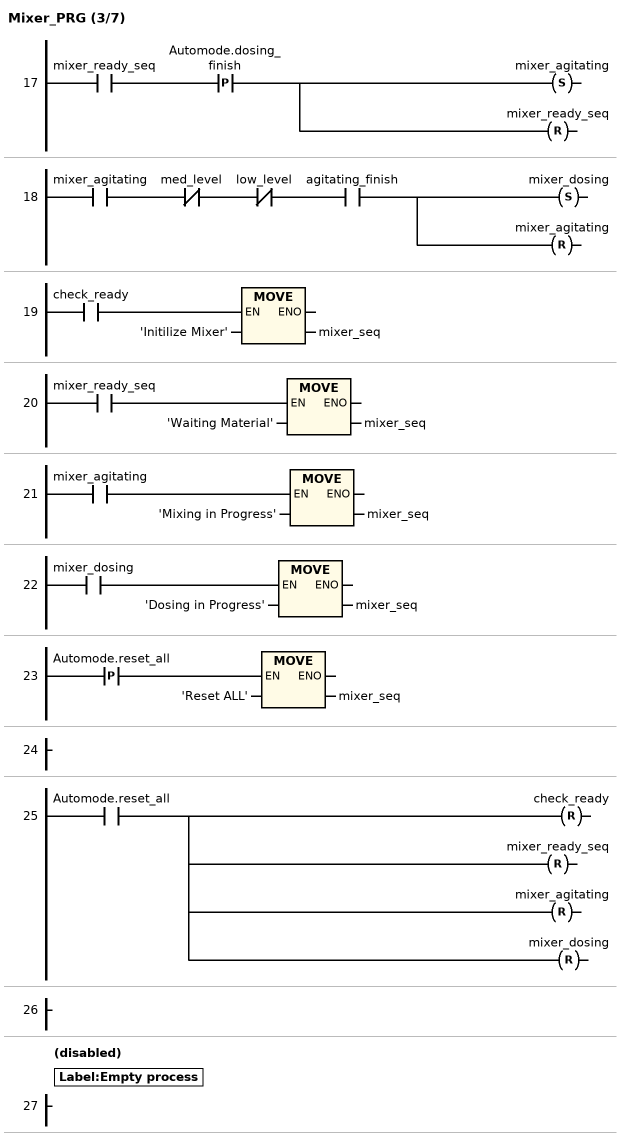
// NETWORK 17
_rt10(CLK := Automode.dosing_finish);
_w3 := mixer_ready_seq AND _rt10.Q;
mixer_agitating S= _w3;
mixer_ready_seq R= _w3;

// NETWORK 18
_w4 := mixer_agitating AND NOT med_level AND NOT low_level AND agitating_finish;
mixer_dosing S= _w4;
mixer_agitating R= _w4;

// NETWORK 19
IF check_ready THEN mixer_seq := 'Initilize Mixer'; END_IF

// NETWORK 20
IF mixer_ready_seq THEN mixer_seq := 'Waiting Material'; END_IF

// NETWORK 21
IF mixer_agitating THEN mixer_seq := 'Mixing in Progress'; END_IF

// NETWORK 22
IF mixer_dosing THEN mixer_seq := 'Dosing in Progress'; END_IF

// NETWORK 23
_rt11(CLK := Automode.reset_all);
IF _rt11.Q THEN mixer_seq := 'Reset ALL'; END_IF

// NETWORK 24

// NETWORK 25
check_ready R= Automode.reset_all;
mixer_ready_seq R= Automode.reset_all;
mixer_agitating R= Automode.reset_all;
mixer_dosing R= Automode.reset_all;

// NETWORK 26

// NETWORK 27 (disabled)
// label: Label:Empty process

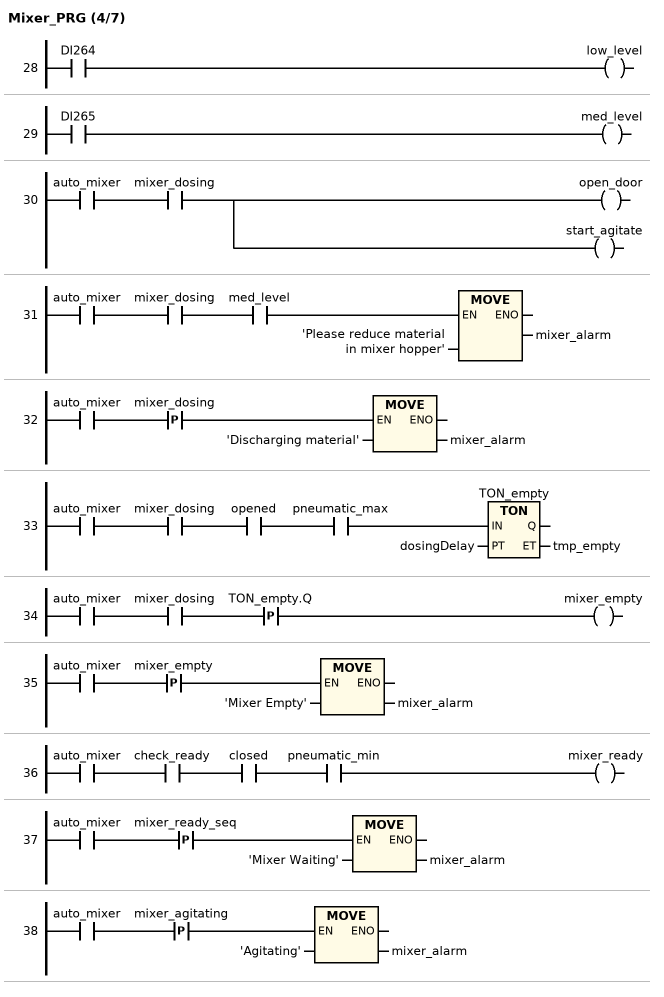
// NETWORK 28
low_level := DI264;

// NETWORK 29
med_level := DI265;

// NETWORK 30
_w5 := auto_mixer AND mixer_dosing;
open_door := _w5;
start_agitate := _w5;

// NETWORK 31
IF auto_mixer AND mixer_dosing AND med_level THEN mixer_alarm := 'Please reduce material in mixer hopper'; END_IF

// NETWORK 32
_rt12(CLK := mixer_dosing);
IF auto_mixer AND _rt12.Q THEN mixer_alarm := 'Discharging material'; END_IF

// NETWORK 33
TON_empty(IN := auto_mixer AND mixer_dosing AND opened AND pneumatic_max, PT := dosingDelay, ET => tmp_empty); // TON

// NETWORK 34
_rt13(CLK := TON_empty.Q);
mixer_empty := auto_mixer AND mixer_dosing AND _rt13.Q;

// NETWORK 35
_rt14(CLK := mixer_empty);
IF auto_mixer AND _rt14.Q THEN mixer_alarm := 'Mixer Empty'; END_IF

// NETWORK 36
mixer_ready := auto_mixer AND check_ready AND closed AND pneumatic_min;

// NETWORK 37
_rt15(CLK := mixer_ready_seq);
IF auto_mixer AND _rt15.Q THEN mixer_alarm := 'Mixer Waiting'; END_IF

// NETWORK 38
_rt16(CLK := mixer_agitating);
IF auto_mixer AND _rt16.Q THEN mixer_alarm := 'Agitating'; END_IF

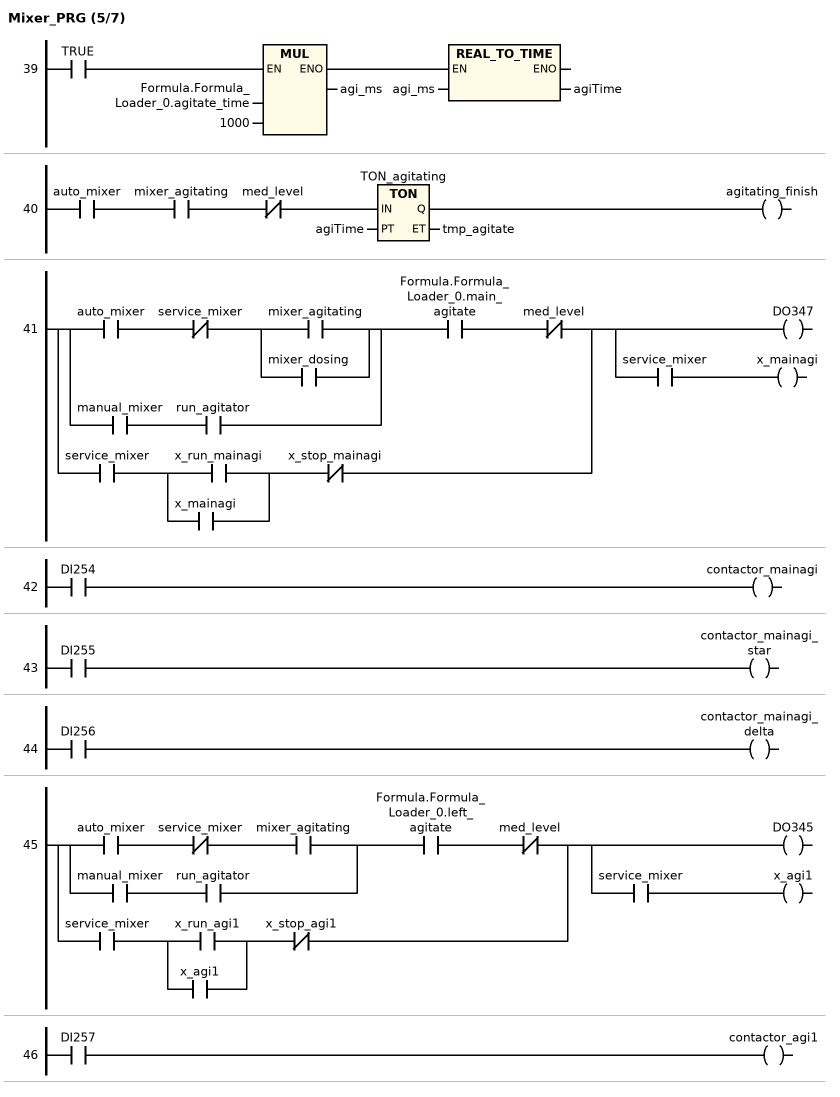
// NETWORK 39
agi_ms := Formula.Formula_Loader_0.agitate_time * 1000;
agiTime := REAL_TO_TIME(agi_ms);

// NETWORK 40
TON_agitating(IN := auto_mixer AND mixer_agitating AND NOT med_level, PT := agiTime, ET => tmp_agitate); // TON
agitating_finish := TON_agitating.Q;

// NETWORK 41
_w6 := (auto_mixer AND NOT service_mixer AND (mixer_agitating OR mixer_dosing) OR manual_mixer AND run_agitator) AND Formula.Formula_Loader_0.main_agitate AND NOT med_level OR service_mixer AND (x_run_mainagi OR x_mainagi) AND NOT x_stop_mainagi;
DO347 := _w6;
x_mainagi := _w6 AND service_mixer;

// NETWORK 42
contactor_mainagi := DI254;

// NETWORK 43
contactor_mainagi_star := DI255;

// NETWORK 44
contactor_mainagi_delta := DI256;

// NETWORK 45
_w7 := (auto_mixer AND NOT service_mixer AND mixer_agitating OR manual_mixer AND run_agitator) AND Formula.Formula_Loader_0.left_agitate AND NOT med_level OR service_mixer AND (x_run_agi1 OR x_agi1) AND NOT x_stop_agi1;
DO345 := _w7;
x_agi1 := _w7 AND service_mixer;

// NETWORK 46
contactor_agi1 := DI257;

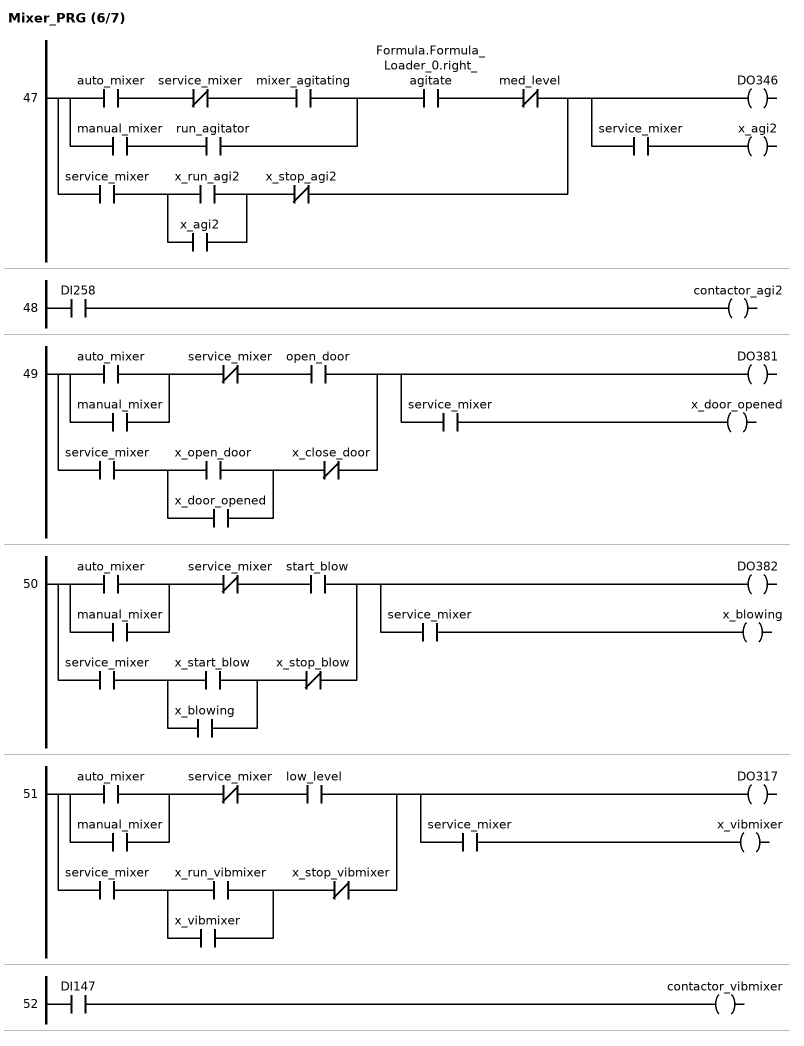
// NETWORK 47
_w8 := (auto_mixer AND NOT service_mixer AND mixer_agitating OR manual_mixer AND run_agitator) AND Formula.Formula_Loader_0.right_agitate AND NOT med_level OR service_mixer AND (x_run_agi2 OR x_agi2) AND NOT x_stop_agi2;
DO346 := _w8;
x_agi2 := _w8 AND service_mixer;

// NETWORK 48
contactor_agi2 := DI258;

// NETWORK 49
_w9 := (auto_mixer OR manual_mixer) AND NOT service_mixer AND open_door OR service_mixer AND (x_open_door OR x_door_opened) AND NOT x_close_door;
DO381 := _w9;
x_door_opened := _w9 AND service_mixer;

// NETWORK 50
_w10 := (auto_mixer OR manual_mixer) AND NOT service_mixer AND start_blow OR service_mixer AND (x_start_blow OR x_blowing) AND NOT x_stop_blow;
DO382 := _w10;
x_blowing := _w10 AND service_mixer;

// NETWORK 51
_w11 := (auto_mixer OR manual_mixer) AND NOT service_mixer AND low_level OR service_mixer AND (x_run_vibmixer OR x_vibmixer) AND NOT x_stop_vibmixer;
DO317 := _w11;
x_vibmixer := _w11 AND service_mixer;

// NETWORK 52
contactor_vibmixer := DI147;

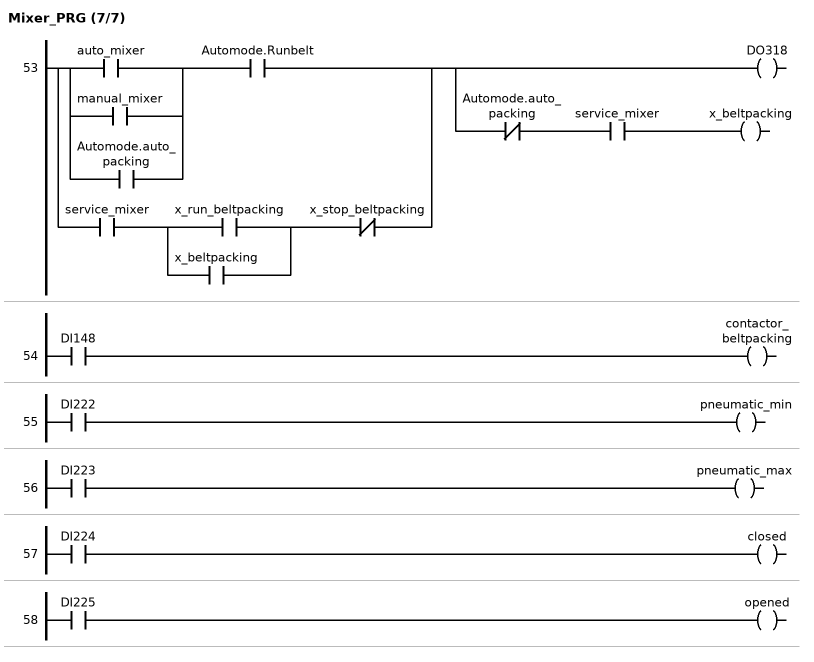
// NETWORK 53
_w12 := (auto_mixer OR manual_mixer OR Automode.auto_packing) AND Automode.Runbelt OR service_mixer AND (x_run_beltpacking OR x_beltpacking) AND NOT x_stop_beltpacking;
DO318 := _w12;
x_beltpacking := _w12 AND NOT Automode.auto_packing AND service_mixer;

// NETWORK 54
contactor_beltpacking := DI148;

// NETWORK 55
pneumatic_min := DI222;

// NETWORK 56
pneumatic_max := DI223;

// NETWORK 57
closed := DI224;

// NETWORK 58
opened := DI225;

END_PROGRAM

// Device/Application/LimeSand
PROGRAM LimeSand
VAR
	auto_lime: BOOL;
	manual_lime: BOOL;
	manual_dosing: BOOL;
	ParamAdjust_bufferlenght: ParamAdjust;
	// meter
	bufferlenght: REAL := 8;
	add_bufferlenght: BOOL;
	sub_bufferlenght: BOOL;
	ParamAdjust_bufferspeed: ParamAdjust;
	// Hz
	bufferspeed: REAL := 20;
	add_bufferspeed: BOOL;
	sub_bufferspeed: BOOL;
	ParamAdjust_beltspeed: ParamAdjust;
	beltspeed: REAL := 0.3;
	add_beltspeed: BOOL;
	sub_beltspeed: BOOL;
	buffering_duration: REAL;
	start_batch: BOOL;
	lime_looper: BOOL;
	finish_dosing: BOOL;
	BAYKON_lime: BAYKON;
	baykon_system: STRING;
	baykon_data: STRING;
	lime_weight: REAL;
	ParamAdjust_LimitLime: ParamAdjust;
	// kg
	limitlime: REAL := 400;
	add_limitlime: BOOL;
	sub_limitlime: BOOL;
	limit_warning: REAL;
	// to HD alarm
	limit_alarm: BOOL;
	limit_alarm_blink: BOOL;
	limit_alarm_hold: BOOL;
	limit_alarm_off: BOOL;
	// from sel switch
	interupted: BOOL;
	start_filling: BOOL;
	filling_request: BOOL;
	tank_filled: BOOL;
	lime_alarm: STRING;
	ready_to_buffer: BOOL;
	getting_lime_weight: BOOL;
	lime_captured: BOOL;
	Constancheck_Lime: Constancheck;
	ParamAdjust_Limeconstant: ParamAdjust;
	// kg
	limeconstant: REAL := 1;
	add_limeconstant: BOOL;
	sub_limeconstant: BOOL;
	lime_stable: BOOL;
	lime_weight_before: REAL;
	filling_ind_blink: BOOL;
	ready_to_fill: BOOL;
	filling_ind_on: BOOL;
	wait_for_fill: BOOL;
	lime_filled: BOOL;
	getting_limeafter: BOOL;
	re_check_lime: BOOL;
	buffering: BOOL;
	lime_starting: REAL;
	buffered: BOOL;
	lime_progress: REAL;
	screw_speed_lime: screw_speed;
	auto_screw_Hz: REAL;
	lime_targetfix: REAL;
	ParamAdjust_maxscrew: ParamAdjust;
	// Hz
	maxscrew: REAL := 40;
	add_maxscrew: BOOL;
	sub_maxscrew: BOOL;
	ParamAdjust_minscrew: ParamAdjust;
	// Hz
	minscrew: REAL := 10;
	add_minscrew: BOOL;
	sub_minscrew: BOOL;
	ParamAdjust_slowscrew: ParamAdjust;
	// %
	slowscrew: REAL := 95;
	add_slowscrew: BOOL;
	sub_slowscrew: BOOL;
	ParamAdjust_slow2screw: ParamAdjust;
	// %
	slow2screw: REAL := 99;
	add_slow2screw: BOOL;
	sub_slow2screw: BOOL;
	run_screw: BOOL;
	finish_buffer: BOOL;
	start_vibrating: BOOL;
	run_vib: BOOL;
	ParamAdjust_vib: ParamAdjust;
	vibreal: REAL := 10;
	add_vibreal: BOOL;
	sub_vibreal: BOOL;
	vibtime: TIME;
	TON_vib: TON;
	tmp_vib: TIME;
	vib_run: BOOL;
	manual_vibration: BOOL;
	end_vibrating: BOOL;
	recheck_lime: BOOL;
	lime_cyclefin: BOOL;
	wait_for_clear: BOOL;
	clear_finish: BOOL;
	finish_button: BOOL;
	cleaning_belt: BOOL;
	manual_clean: BOOL;
	TON_clean: TON;
	cleaning_duration: REAL;
	bufferingtime: TIME;
	cleaningtime: TIME;
	tmp_clean: TIME;
	cleared: BOOL;
	run_belt: BOOL;
	high_speed: BOOL;
	buffer_button: BOOL;
	buffer_belt: BOOL;
	slow_speed: BOOL;
	TON_buffer: TON;
	tmp_buffer: TIME;
	service_lime: BOOL := true;
	run_viblime: BOOL;
	x_run_viblime: BOOL;
	x_stop_viblime: BOOL;
	x_viblime: BOOL;
	run_vibsand: BOOL;
	x_vibsand: BOOL;
	x_run_vibsand: BOOL;
	x_stop_vibsand: BOOL;
	INVT_AO_screwlime: INVT_AO;
	x_screwlime: BOOL;
	screw_fwd: BOOL;
	screw_run: BOOL;
	screw_standby: BOOL;
	screw_rvs: BOOL;
	rvs_relay: BOOL;
	screw_fault: BOOL;
	screw_Hz: REAL;
	x_run_screw: BOOL;
	x_stop_screw: BOOL;
	ParamAdjust_limeservice: ParamAdjust;
	screw_service: REAL := 20;
	add_screwservice: BOOL;
	sub_screwservice: BOOL;
	ParamAdjust_beltservice: ParamAdjust;
	belt_service: REAL := 20;
	add_beltservice: BOOL;
	sub_beltservice: BOOL;
	auto_belt_Hz: REAL;
	belt_Hz: REAL := 20;
	INVT_AO_belt: INVT_AO;
	x_belt: BOOL;
	belt_fwd: BOOL;
	belt_run: BOOL;
	belt_standby: BOOL;
	belt_rvs: BOOL;
	b_relay: BOOL;
	belt_fault: BOOL;
	x_run_belt: BOOL;
	x_stop_belt: BOOL;
	auto_limex: BOOL;
	manual_limex: BOOL;
	service_limex: BOOL;
	contactor_viblime: BOOL;
	contactor_vibsand: BOOL;
	contactor_screwlime: BOOL;
	contactor_belt: BOOL;
	dosing_ready: BOOL;
	fast_belt: BOOL;
	dosing_finish: BOOL;
	open_valve: BOOL;
	filling_ind_blink2: BOOL;
	lime_ready: BOOL;
	// from button
	start_buffer: BOOL;
	TON_delay_lime: TON;
	ParamAdjust_limeelaay: ParamAdjust;
	// s
	limedelay: REAL := 3;
	add_limedelay: BOOL;
	sub_limedelay: BOOL;
	limedelayms: REAL;
	limedelayTime: TIME;
	tmp_limeedelay: TIME;
	ParamAdjust_fastspeed: ParamAdjust;
	// Hz
	cleanspeed: REAL := 50;
	add_cleanspeed: BOOL;
	sub_cleanspeed: BOOL;
	buffer_coef: REAL;
	buffering_time: REAL;
	fast_speed: BOOL;
	run_belt2: BOOL;
	run_screw2: BOOL;
	vibrealms: REAL;
	lime_finish: BOOL;
	belt_clearup: BOOL;
	run_limescrew: BOOL;
	run_sandbelt: BOOL;
	sand_opened: BOOL;
	x_valve: BOOL;
	x_open_valve: BOOL;
	x_close_valve: BOOL;
	bufferingtimex: REAL;
	sand_closed: BOOL;
	manual_weight: BOOL;
	checking_seq: BOOL;
	LimeSand_ready: BOOL;
	waiting_mixer: BOOL;
	buffering_seq: BOOL;
	buffering_finish: BOOL;
	dosing_seq: BOOL;
	lime_finish_seq: BOOL;
	clean_seq: BOOL;
	lime_a: REAL;
	lime_amp: REAL;
	belt_a: REAL;
	belt_amp: REAL;
	start_lime: REAL;
	end_lime: REAL;
	weighting_time: INT;
	weighting_duration: INT;
	m_lime_start: BOOL;
	m_lime_stop: BOOL;
	manual_liming: BOOL;
	m_run_belt: BOOL;
	m_start_lime: REAL;
	m_lime_progress: REAL;
	m_lime_finish: BOOL;
	TON_liming: TON;
	tmp_liming: TIME;
	m_run_screw: BOOL;
	lime_seq: STRING;
	param_clean: INT;
	ParamAdjust_clear: ParamAdjust;
	// second
	clear_param: REAL := 15;
	add_clear: BOOL;
	sub_clear: BOOL;
	baykon_mati: BOOL;
	TON_mati: TON;
	tmpmati: TIME;
	baykon_disconnect: BOOL;
	baykon_dis: BOOL;
	TON_murub: TON;
	tmpmurub: TIME;
END_VAR
VAR // added by the converter: edge detectors and wires of the graphical bodies
    _rt1, _rt2, _rt3, _rt4, _rt5, _rt6, _rt7, _rt8, _rt9, _rt10, _rt11, _rt12, _rt13, _rt14, _rt15, _rt16, _rt17, _rt18, _rt19 : R_TRIG;
    _w1, _w2, _w3, _w4, _w5, _w6, _w7, _w8, _w9, _w10, _w11, _w12, _w13, _w14, _w15 : BOOL;
    _ft1 : F_TRIG;
END_VAR

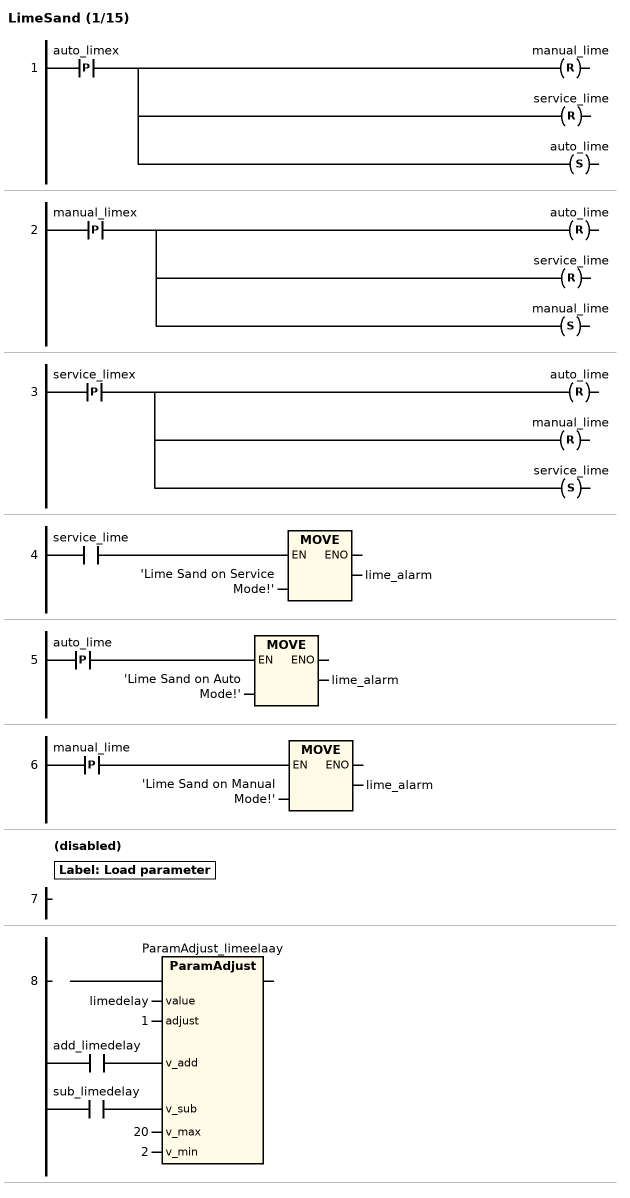
// NETWORK 1
_rt1(CLK := auto_limex);
manual_lime R= _rt1.Q;
service_lime R= _rt1.Q;
auto_lime S= _rt1.Q;

// NETWORK 2
_rt2(CLK := manual_limex);
auto_lime R= _rt2.Q;
service_lime R= _rt2.Q;
manual_lime S= _rt2.Q;

// NETWORK 3
_rt3(CLK := service_limex);
auto_lime R= _rt3.Q;
manual_lime R= _rt3.Q;
service_lime S= _rt3.Q;

// NETWORK 4
IF service_lime THEN lime_alarm := 'Lime Sand on Service Mode!'; END_IF

// NETWORK 5
_rt4(CLK := auto_lime);
IF _rt4.Q THEN lime_alarm := 'Lime Sand on Auto Mode!'; END_IF

// NETWORK 6
_rt5(CLK := manual_lime);
IF _rt5.Q THEN lime_alarm := 'Lime Sand on Manual Mode!'; END_IF

// NETWORK 7 (disabled)
// label: Label: Load parameter

// NETWORK 8
ParamAdjust_limeelaay(
    value := limedelay,
    adjust := 1,
    v_add := add_limedelay,
    v_sub := sub_limedelay,
    v_max := 20,
    v_min := 2); // ParamAdjust

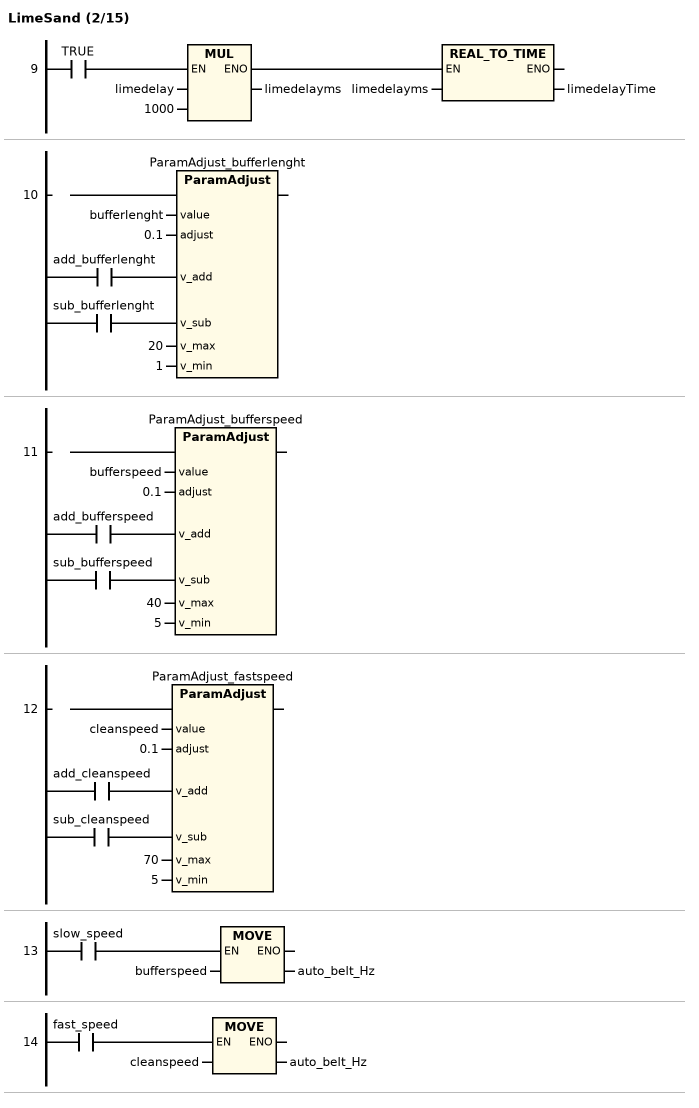
// NETWORK 9
limedelayms := limedelay * 1000;
limedelayTime := REAL_TO_TIME(limedelayms);

// NETWORK 10
ParamAdjust_bufferlenght(
    value := bufferlenght,
    adjust := 0.1,
    v_add := add_bufferlenght,
    v_sub := sub_bufferlenght,
    v_max := 20,
    v_min := 1); // ParamAdjust

// NETWORK 11
ParamAdjust_bufferspeed(
    value := bufferspeed,
    adjust := 0.1,
    v_add := add_bufferspeed,
    v_sub := sub_bufferspeed,
    v_max := 40,
    v_min := 5); // ParamAdjust

// NETWORK 12
ParamAdjust_fastspeed(
    value := cleanspeed,
    adjust := 0.1,
    v_add := add_cleanspeed,
    v_sub := sub_cleanspeed,
    v_max := 70,
    v_min := 5); // ParamAdjust

// NETWORK 13
IF slow_speed THEN auto_belt_Hz := bufferspeed; END_IF

// NETWORK 14
IF fast_speed THEN auto_belt_Hz := cleanspeed; END_IF

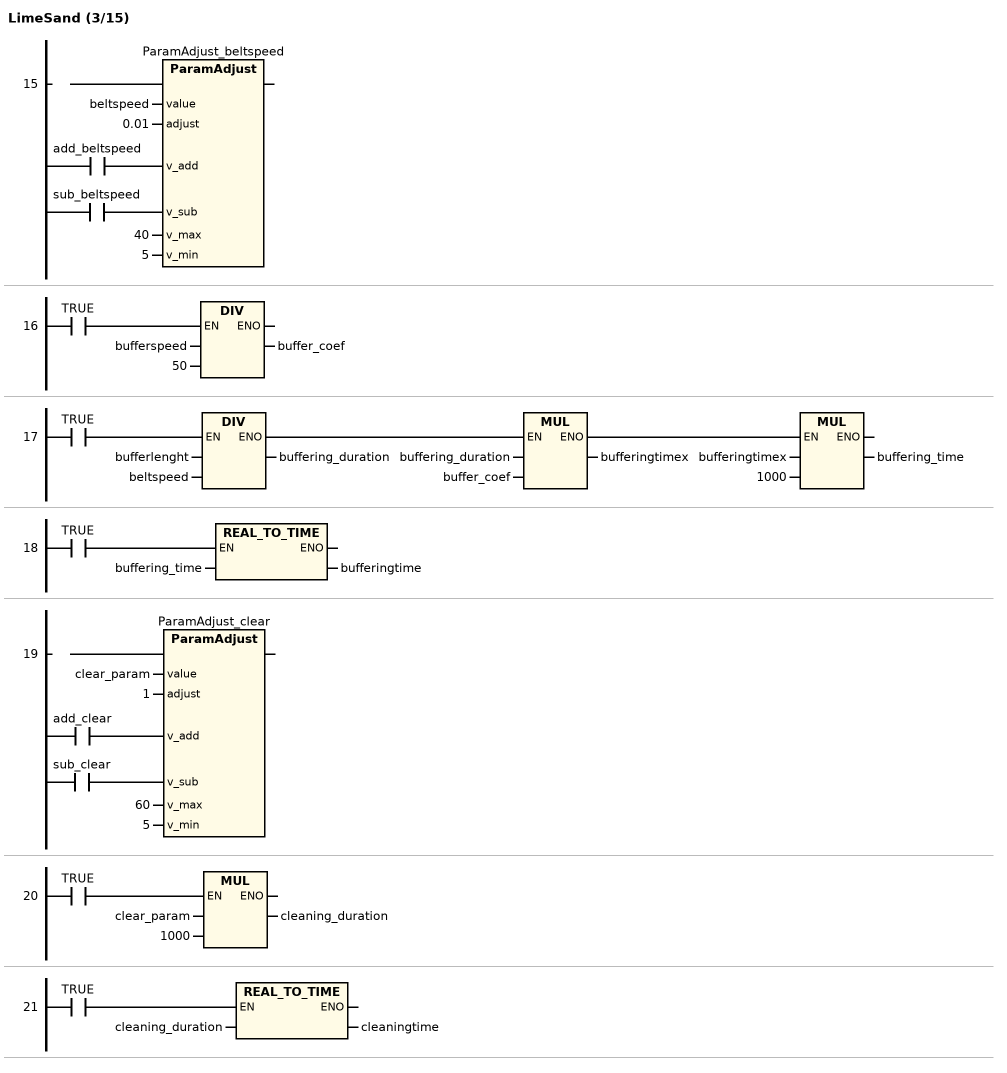
// NETWORK 15
ParamAdjust_beltspeed(
    value := beltspeed,
    adjust := 0.01,
    v_add := add_beltspeed,
    v_sub := sub_beltspeed,
    v_max := 40,
    v_min := 5); // ParamAdjust

// NETWORK 16
buffer_coef := bufferspeed / 50;

// NETWORK 17
buffering_duration := bufferlenght / beltspeed;
bufferingtimex := buffering_duration * buffer_coef;
buffering_time := bufferingtimex * 1000;

// NETWORK 18
bufferingtime := REAL_TO_TIME(buffering_time);

// NETWORK 19
ParamAdjust_clear(
    value := clear_param,
    adjust := 1,
    v_add := add_clear,
    v_sub := sub_clear,
    v_max := 60,
    v_min := 5); // ParamAdjust

// NETWORK 20
cleaning_duration := clear_param * 1000;

// NETWORK 21
cleaningtime := REAL_TO_TIME(cleaning_duration);

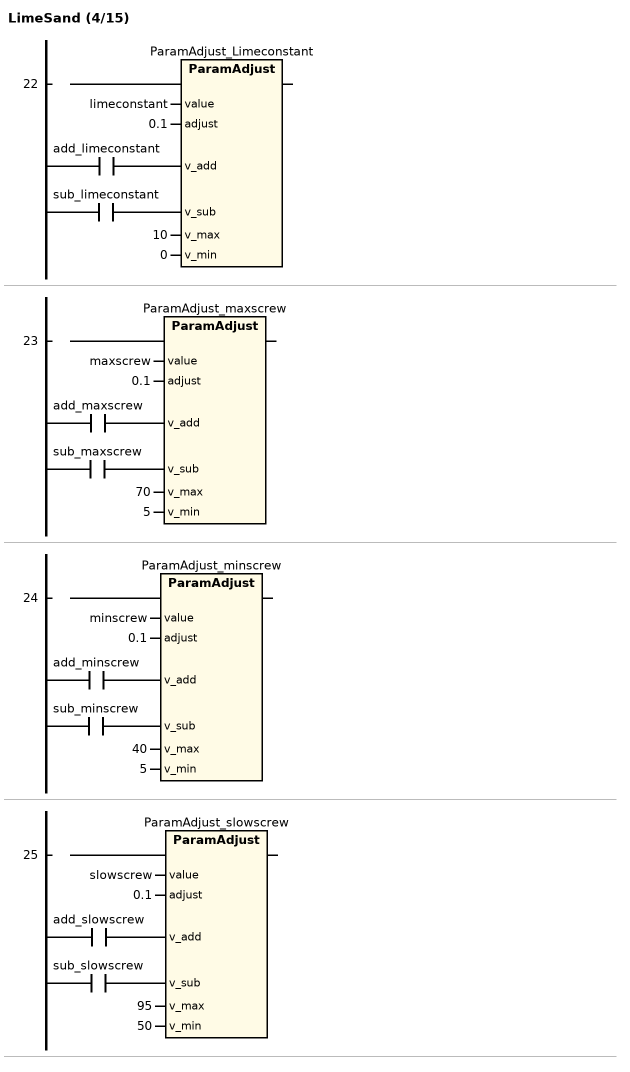
// NETWORK 22
ParamAdjust_Limeconstant(
    value := limeconstant,
    adjust := 0.1,
    v_add := add_limeconstant,
    v_sub := sub_limeconstant,
    v_max := 10,
    v_min := 0); // ParamAdjust

// NETWORK 23
ParamAdjust_maxscrew(
    value := maxscrew,
    adjust := 0.1,
    v_add := add_maxscrew,
    v_sub := sub_maxscrew,
    v_max := 70,
    v_min := 5); // ParamAdjust

// NETWORK 24
ParamAdjust_minscrew(
    value := minscrew,
    adjust := 0.1,
    v_add := add_minscrew,
    v_sub := sub_minscrew,
    v_max := 40,
    v_min := 5); // ParamAdjust

// NETWORK 25
ParamAdjust_slowscrew(
    value := slowscrew,
    adjust := 0.1,
    v_add := add_slowscrew,
    v_sub := sub_slowscrew,
    v_max := 95,
    v_min := 50); // ParamAdjust

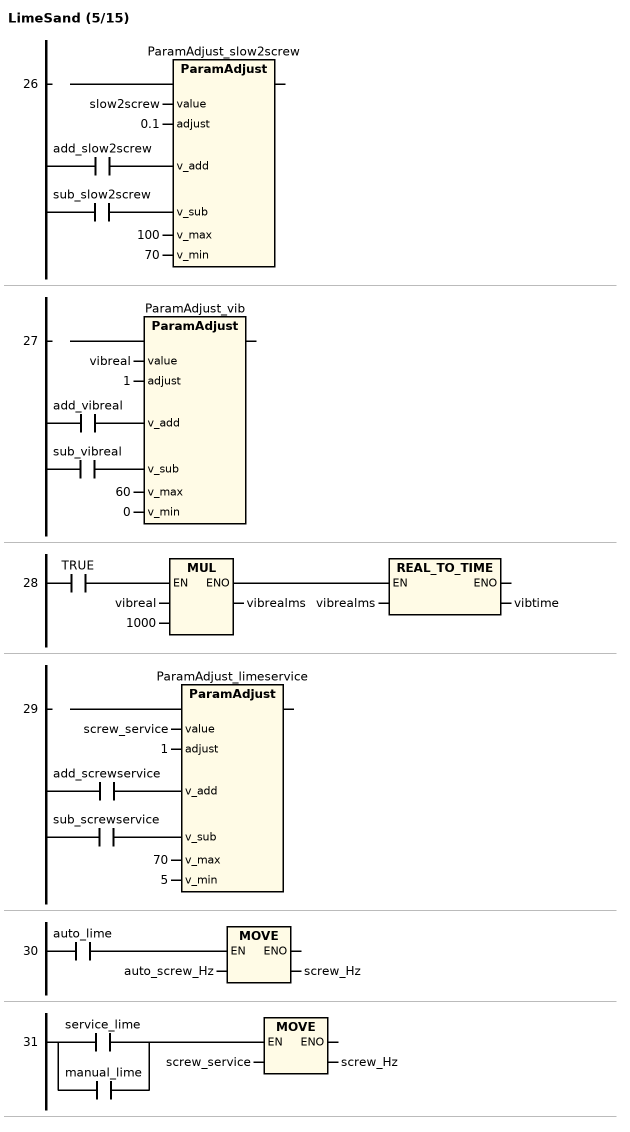
// NETWORK 26
ParamAdjust_slow2screw(
    value := slow2screw,
    adjust := 0.1,
    v_add := add_slow2screw,
    v_sub := sub_slow2screw,
    v_max := 100,
    v_min := 70); // ParamAdjust

// NETWORK 27
ParamAdjust_vib(
    value := vibreal,
    adjust := 1,
    v_add := add_vibreal,
    v_sub := sub_vibreal,
    v_max := 60,
    v_min := 0); // ParamAdjust

// NETWORK 28
vibrealms := vibreal * 1000;
vibtime := REAL_TO_TIME(vibrealms);

// NETWORK 29
ParamAdjust_limeservice(
    value := screw_service,
    adjust := 1,
    v_add := add_screwservice,
    v_sub := sub_screwservice,
    v_max := 70,
    v_min := 5); // ParamAdjust

// NETWORK 30
IF auto_lime THEN screw_Hz := auto_screw_Hz; END_IF

// NETWORK 31
IF service_lime OR manual_lime THEN screw_Hz := screw_service; END_IF

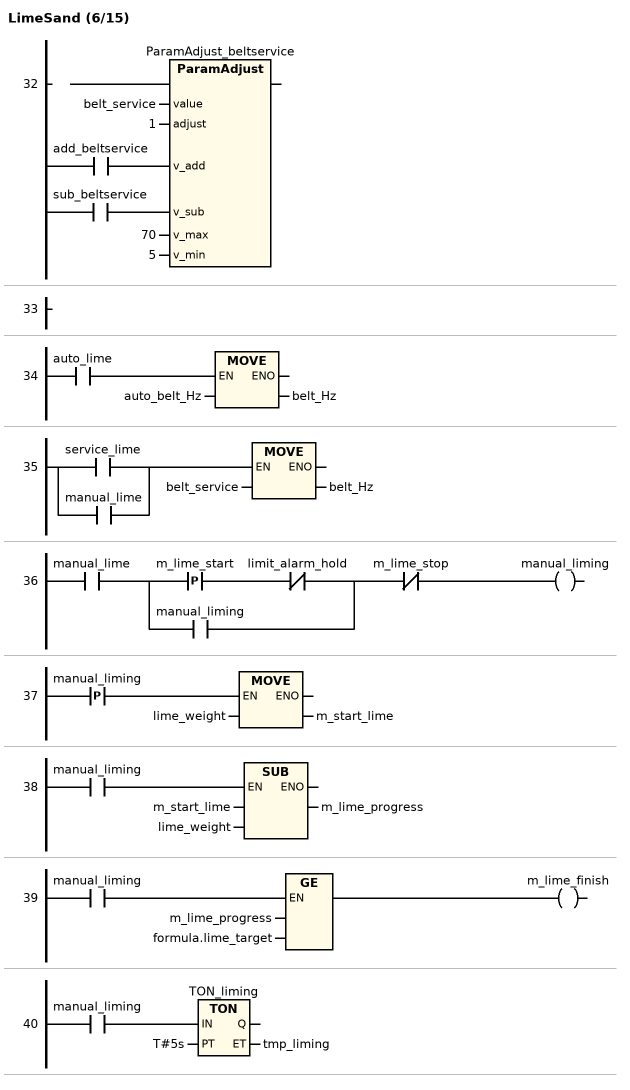
// NETWORK 32
ParamAdjust_beltservice(
    value := belt_service,
    adjust := 1,
    v_add := add_beltservice,
    v_sub := sub_beltservice,
    v_max := 70,
    v_min := 5); // ParamAdjust

// NETWORK 33

// NETWORK 34
IF auto_lime THEN belt_Hz := auto_belt_Hz; END_IF

// NETWORK 35
IF service_lime OR manual_lime THEN belt_Hz := belt_service; END_IF

// NETWORK 36
_rt6(CLK := m_lime_start);
manual_liming := manual_lime AND (_rt6.Q AND NOT limit_alarm_hold OR manual_liming) AND NOT m_lime_stop;

// NETWORK 37
_rt7(CLK := manual_liming);
IF _rt7.Q THEN m_start_lime := lime_weight; END_IF

// NETWORK 38
IF manual_liming THEN m_lime_progress := m_start_lime - lime_weight; END_IF

// NETWORK 39
m_lime_finish := manual_liming AND m_lime_progress >= formula.lime_target;

// NETWORK 40
TON_liming(IN := manual_liming, PT := T#5s, ET => tmp_liming); // TON

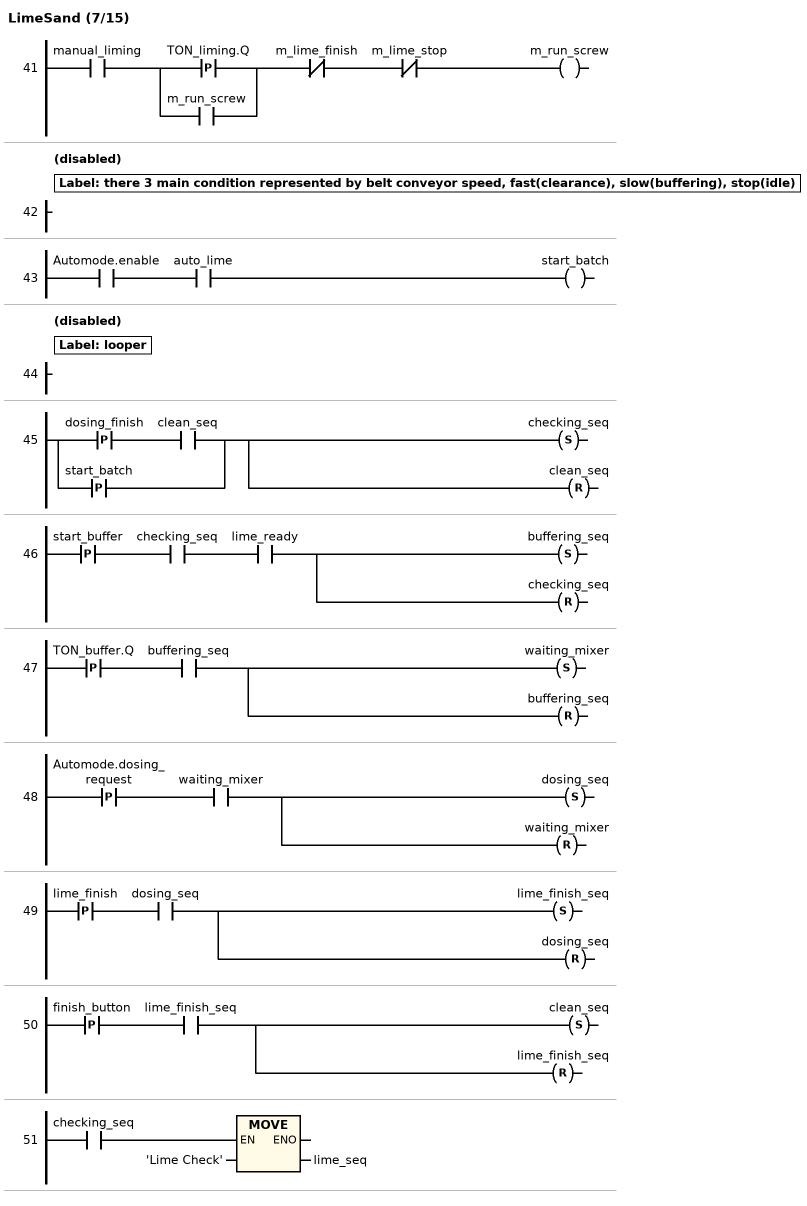
// NETWORK 41
_rt8(CLK := TON_liming.Q);
m_run_screw := manual_liming AND (_rt8.Q OR m_run_screw) AND NOT m_lime_finish AND NOT m_lime_stop;

// NETWORK 42 (disabled)
// label: Label: there 3 main condition represented by belt conveyor speed, fast(clearance), slow(buffering), stop(idle)

// NETWORK 43
start_batch := Automode.enable AND auto_lime;

// NETWORK 44 (disabled)
// label: Label: looper

// NETWORK 45
_rt9(CLK := dosing_finish);
_rt10(CLK := start_batch);
_w1 := _rt9.Q AND clean_seq OR _rt10.Q;
checking_seq S= _w1;
clean_seq R= _w1;

// NETWORK 46
_rt11(CLK := start_buffer);
_w2 := _rt11.Q AND checking_seq AND lime_ready;
buffering_seq S= _w2;
checking_seq R= _w2;

// NETWORK 47
_rt12(CLK := TON_buffer.Q);
_w3 := _rt12.Q AND buffering_seq;
waiting_mixer S= _w3;
buffering_seq R= _w3;

// NETWORK 48
_rt13(CLK := Automode.dosing_request);
_w4 := _rt13.Q AND waiting_mixer;
dosing_seq S= _w4;
waiting_mixer R= _w4;

// NETWORK 49
_rt14(CLK := lime_finish);
_w5 := _rt14.Q AND dosing_seq;
lime_finish_seq S= _w5;
dosing_seq R= _w5;

// NETWORK 50
_rt15(CLK := finish_button);
_w6 := _rt15.Q AND lime_finish_seq;
clean_seq S= _w6;
lime_finish_seq R= _w6;

// NETWORK 51
IF checking_seq THEN lime_seq := 'Lime Check'; END_IF

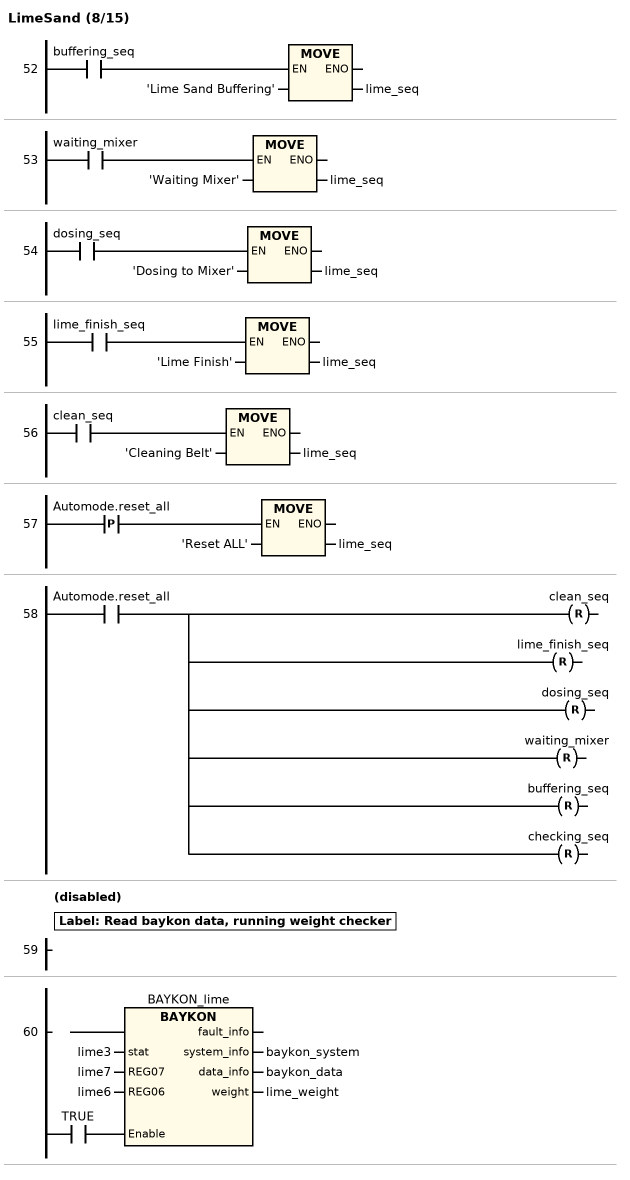
// NETWORK 52
IF buffering_seq THEN lime_seq := 'Lime Sand Buffering'; END_IF

// NETWORK 53
IF waiting_mixer THEN lime_seq := 'Waiting Mixer'; END_IF

// NETWORK 54
IF dosing_seq THEN lime_seq := 'Dosing to Mixer'; END_IF

// NETWORK 55
IF lime_finish_seq THEN lime_seq := 'Lime Finish'; END_IF

// NETWORK 56
IF clean_seq THEN lime_seq := 'Cleaning Belt'; END_IF

// NETWORK 57
_rt16(CLK := Automode.reset_all);
IF _rt16.Q THEN lime_seq := 'Reset ALL'; END_IF

// NETWORK 58
clean_seq R= Automode.reset_all;
lime_finish_seq R= Automode.reset_all;
dosing_seq R= Automode.reset_all;
waiting_mixer R= Automode.reset_all;
buffering_seq R= Automode.reset_all;
checking_seq R= Automode.reset_all;

// NETWORK 59 (disabled)
// label: Label: Read baykon data, running weight checker

// NETWORK 60
BAYKON_lime(
    stat := lime3,
    REG07 := lime7,
    REG06 := lime6,
    Enable := TRUE,
    system_info => baykon_system,
    data_info => baykon_data,
    weight => lime_weight); // BAYKON

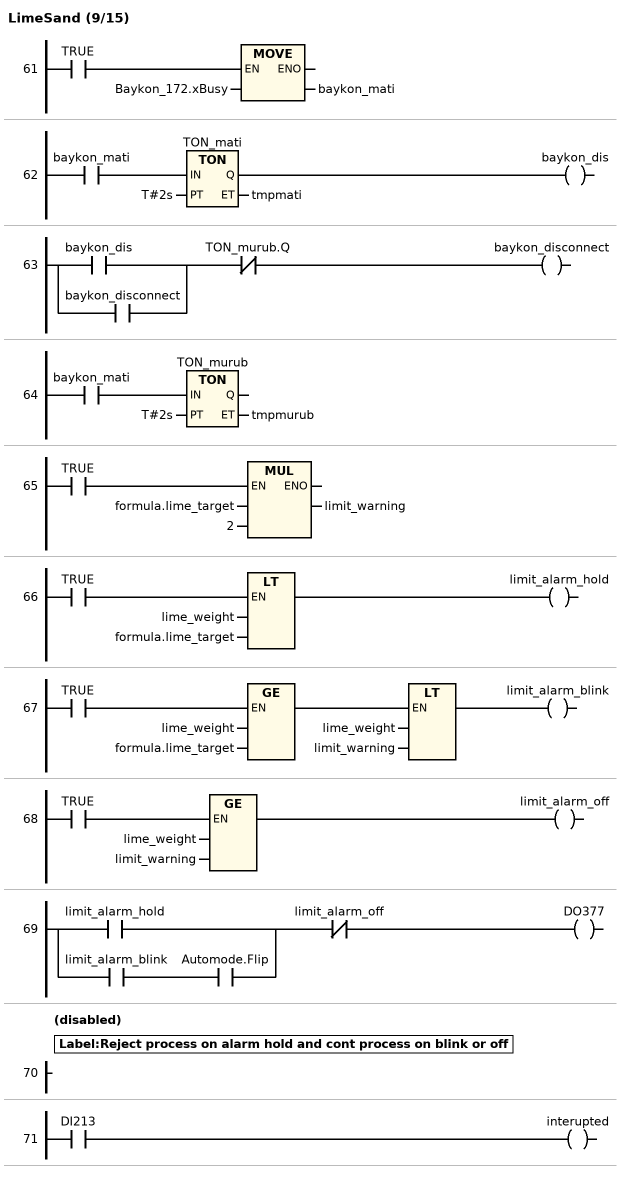
// NETWORK 61
baykon_mati := Baykon_172.xBusy;

// NETWORK 62
TON_mati(IN := baykon_mati, PT := T#2s, ET => tmpmati); // TON
baykon_dis := TON_mati.Q;

// NETWORK 63
baykon_disconnect := (baykon_dis OR baykon_disconnect) AND NOT TON_murub.Q;

// NETWORK 64
TON_murub(IN := baykon_mati, PT := T#2s, ET => tmpmurub); // TON

// NETWORK 65
limit_warning := formula.lime_target * 2;

// NETWORK 66
limit_alarm_hold := lime_weight < formula.lime_target;

// NETWORK 67
limit_alarm_blink := lime_weight >= formula.lime_target AND lime_weight < limit_warning;

// NETWORK 68
limit_alarm_off := lime_weight >= limit_warning;

// NETWORK 69
DO377 := (limit_alarm_hold OR limit_alarm_blink AND Automode.Flip) AND NOT limit_alarm_off;

// NETWORK 70 (disabled)
// label: Label:Reject process on alarm hold and cont process on blink or off

// NETWORK 71
interupted := DI213;

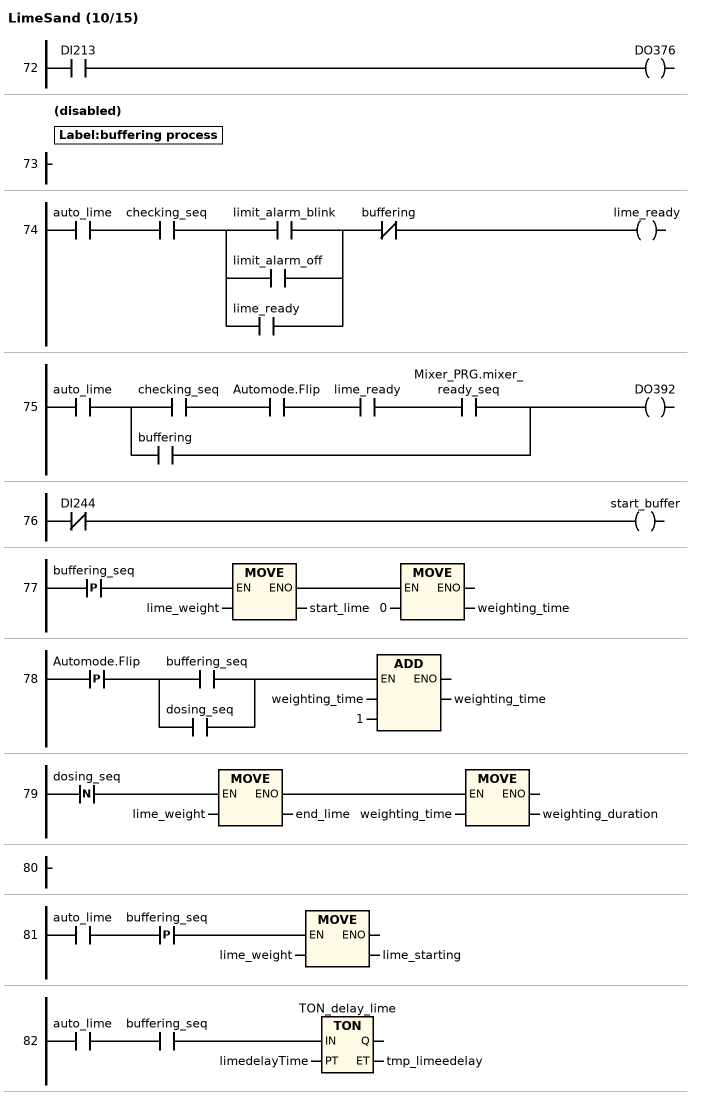
// NETWORK 72
DO376 := DI213;

// NETWORK 73 (disabled)
// label: Label:buffering process

// NETWORK 74
lime_ready := auto_lime AND checking_seq AND (limit_alarm_blink OR limit_alarm_off OR lime_ready) AND NOT buffering;

// NETWORK 75
DO392 := auto_lime AND (checking_seq AND Automode.Flip AND lime_ready AND Mixer_PRG.mixer_ready_seq OR buffering);

// NETWORK 76
start_buffer := NOT DI244;

// NETWORK 77
_rt17(CLK := buffering_seq);
_w7 := _rt17.Q;
IF _w7 THEN start_lime := lime_weight; END_IF
IF _w7 THEN weighting_time := 0; END_IF

// NETWORK 78
_rt18(CLK := Automode.Flip);
IF _rt18.Q AND (buffering_seq OR dosing_seq) THEN weighting_time := weighting_time + 1; END_IF

// NETWORK 79
_ft1(CLK := dosing_seq);
_w8 := _ft1.Q;
IF _w8 THEN end_lime := lime_weight; END_IF
IF _w8 THEN weighting_duration := weighting_time; END_IF

// NETWORK 80

// NETWORK 81
_rt19(CLK := buffering_seq);
IF auto_lime AND _rt19.Q THEN lime_starting := lime_weight; END_IF

// NETWORK 82
TON_delay_lime(IN := auto_lime AND buffering_seq, PT := limedelayTime, ET => tmp_limeedelay); // TON

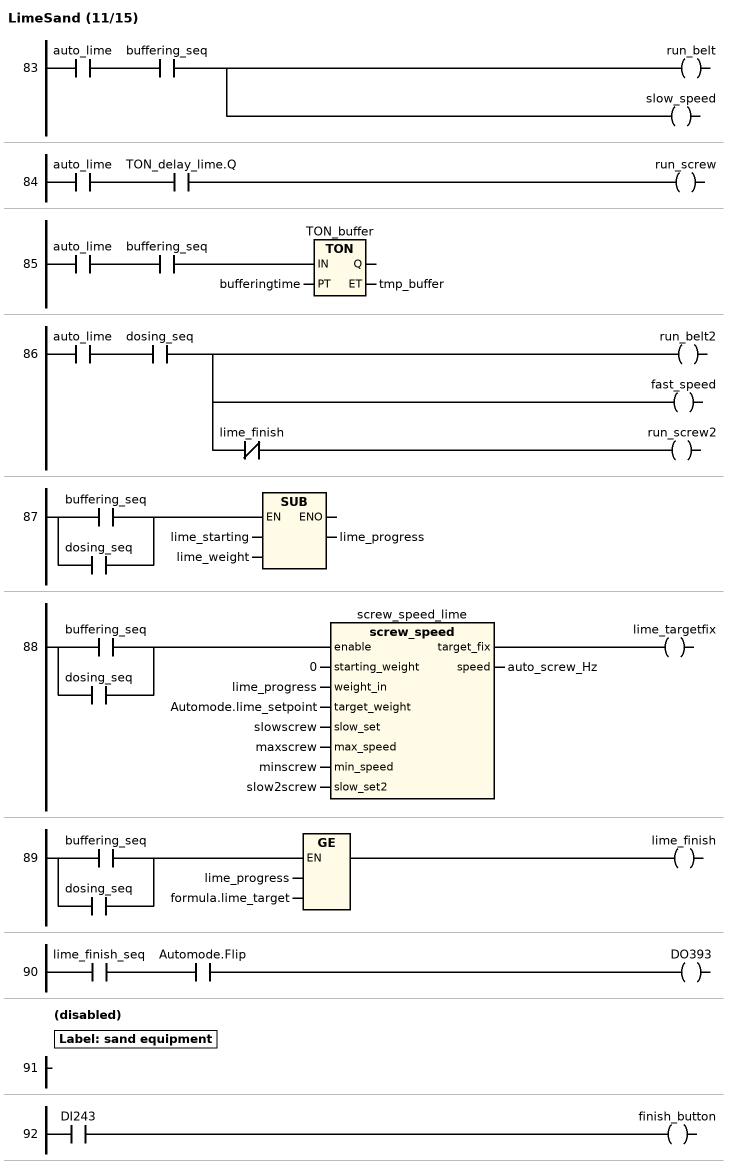
// NETWORK 83
_w9 := auto_lime AND buffering_seq;
run_belt := _w9;
slow_speed := _w9;

// NETWORK 84
run_screw := auto_lime AND TON_delay_lime.Q;

// NETWORK 85
TON_buffer(IN := auto_lime AND buffering_seq, PT := bufferingtime, ET => tmp_buffer); // TON

// NETWORK 86
_w10 := auto_lime AND dosing_seq;
run_belt2 := _w10;
fast_speed := _w10;
run_screw2 := _w10 AND NOT lime_finish;

// NETWORK 87
IF buffering_seq OR dosing_seq THEN lime_progress := lime_starting - lime_weight; END_IF

// NETWORK 88
screw_speed_lime(
    enable := buffering_seq OR dosing_seq,
    starting_weight := 0,
    weight_in := lime_progress,
    target_weight := Automode.lime_setpoint,
    slow_set := slowscrew,
    max_speed := maxscrew,
    min_speed := minscrew,
    slow_set2 := slow2screw,
    speed => auto_screw_Hz); // screw_speed
lime_targetfix := screw_speed_lime.target_fix;

// NETWORK 89
lime_finish := (buffering_seq OR dosing_seq) AND lime_progress >= formula.lime_target;

// NETWORK 90
DO393 := lime_finish_seq AND Automode.Flip;

// NETWORK 91 (disabled)
// label: Label: sand equipment

// NETWORK 92
finish_button := DI243;

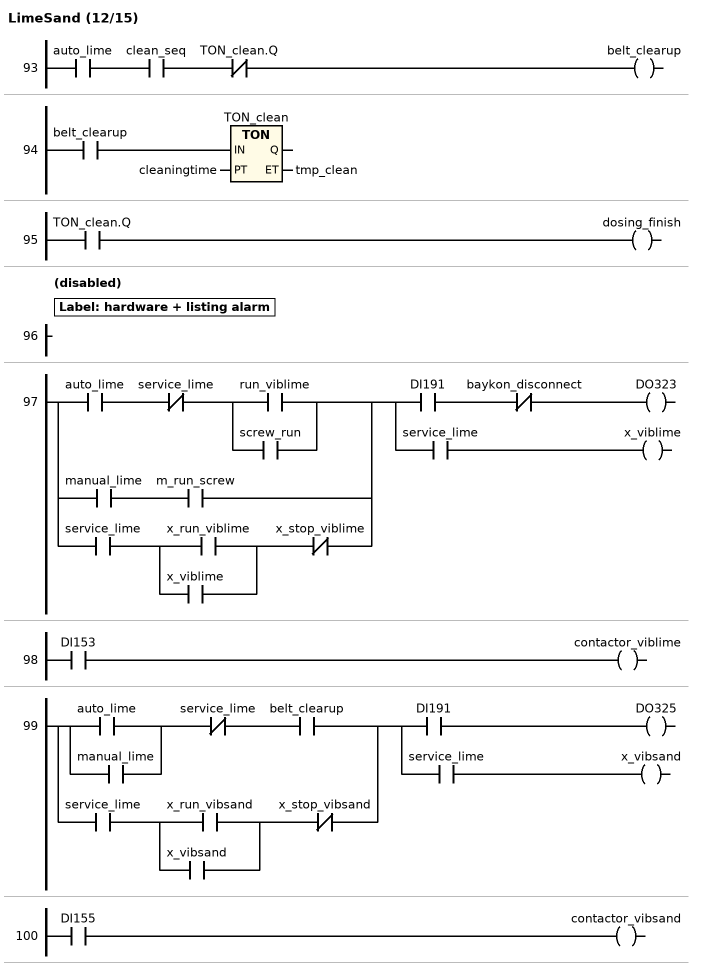
// NETWORK 93
belt_clearup := auto_lime AND clean_seq AND NOT TON_clean.Q;

// NETWORK 94
TON_clean(IN := belt_clearup, PT := cleaningtime, ET => tmp_clean); // TON

// NETWORK 95
dosing_finish := TON_clean.Q;

// NETWORK 96 (disabled)
// label: Label: hardware + listing alarm

// NETWORK 97
_w11 := auto_lime AND NOT service_lime AND (run_viblime OR screw_run) OR manual_lime AND m_run_screw OR service_lime AND (x_run_viblime OR x_viblime) AND NOT x_stop_viblime;
DO323 := _w11 AND DI191 AND NOT baykon_disconnect;
x_viblime := _w11 AND service_lime;

// NETWORK 98
contactor_viblime := DI153;

// NETWORK 99
_w12 := (auto_lime OR manual_lime) AND NOT service_lime AND belt_clearup OR service_lime AND (x_run_vibsand OR x_vibsand) AND NOT x_stop_vibsand;
DO325 := _w12 AND DI191;
x_vibsand := _w12 AND service_lime;

// NETWORK 100
contactor_vibsand := DI155;

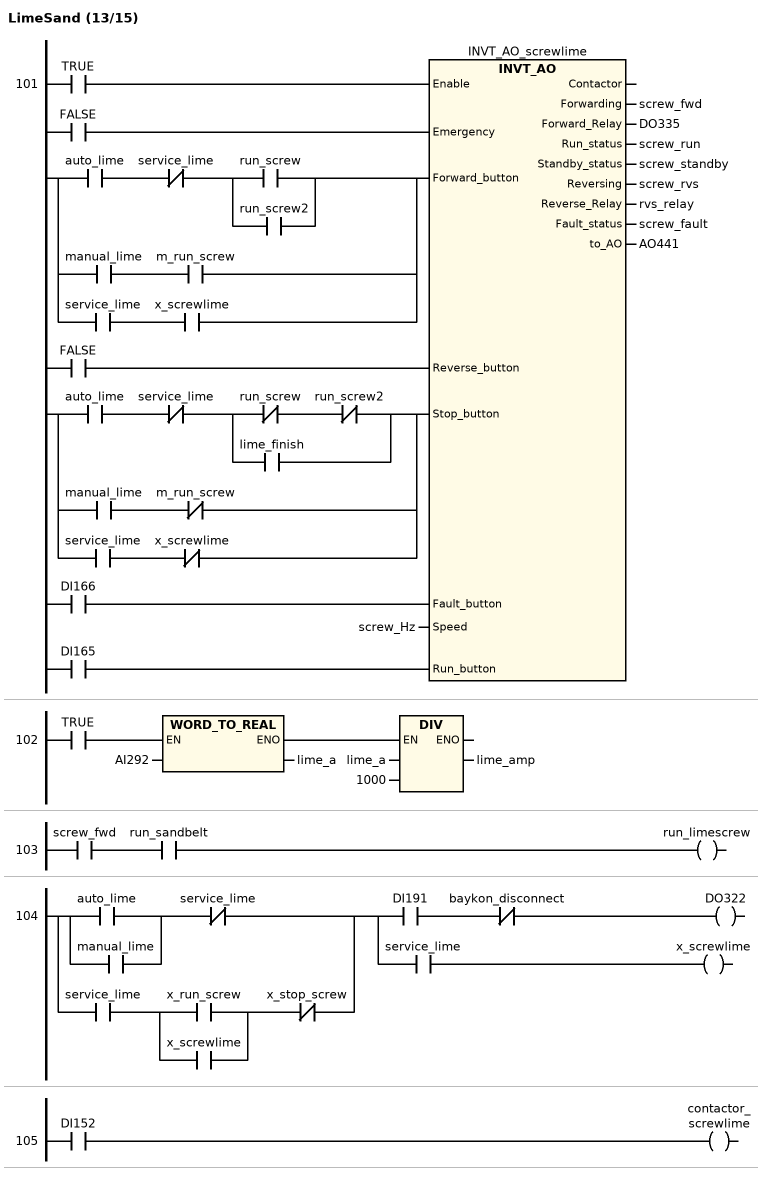
// NETWORK 101
INVT_AO_screwlime(
    Enable := TRUE,
    Emergency := FALSE,
    Forward_button := auto_lime AND NOT service_lime AND (run_screw OR run_screw2) OR manual_lime AND m_run_screw OR service_lime AND x_screwlime,
    Reverse_button := FALSE,
    Stop_button := auto_lime AND NOT service_lime AND (NOT run_screw AND NOT run_screw2 OR lime_finish) OR manual_lime AND NOT m_run_screw OR service_lime AND NOT x_screwlime,
    Fault_button := DI166,
    Speed := screw_Hz,
    Run_button := DI165,
    Forwarding => screw_fwd,
    Forward_Relay => DO335,
    Run_status => screw_run,
    Standby_status => screw_standby,
    Reversing => screw_rvs,
    Reverse_Relay => rvs_relay,
    Fault_status => screw_fault,
    to_AO => AO441); // INVT_AO

// NETWORK 102
lime_a := WORD_TO_REAL(AI292);
lime_amp := lime_a / 1000;

// NETWORK 103
run_limescrew := screw_fwd AND run_sandbelt;

// NETWORK 104
_w13 := (auto_lime OR manual_lime) AND NOT service_lime OR service_lime AND (x_run_screw OR x_screwlime) AND NOT x_stop_screw;
DO322 := _w13 AND DI191 AND NOT baykon_disconnect;
x_screwlime := _w13 AND service_lime;

// NETWORK 105
contactor_screwlime := DI152;

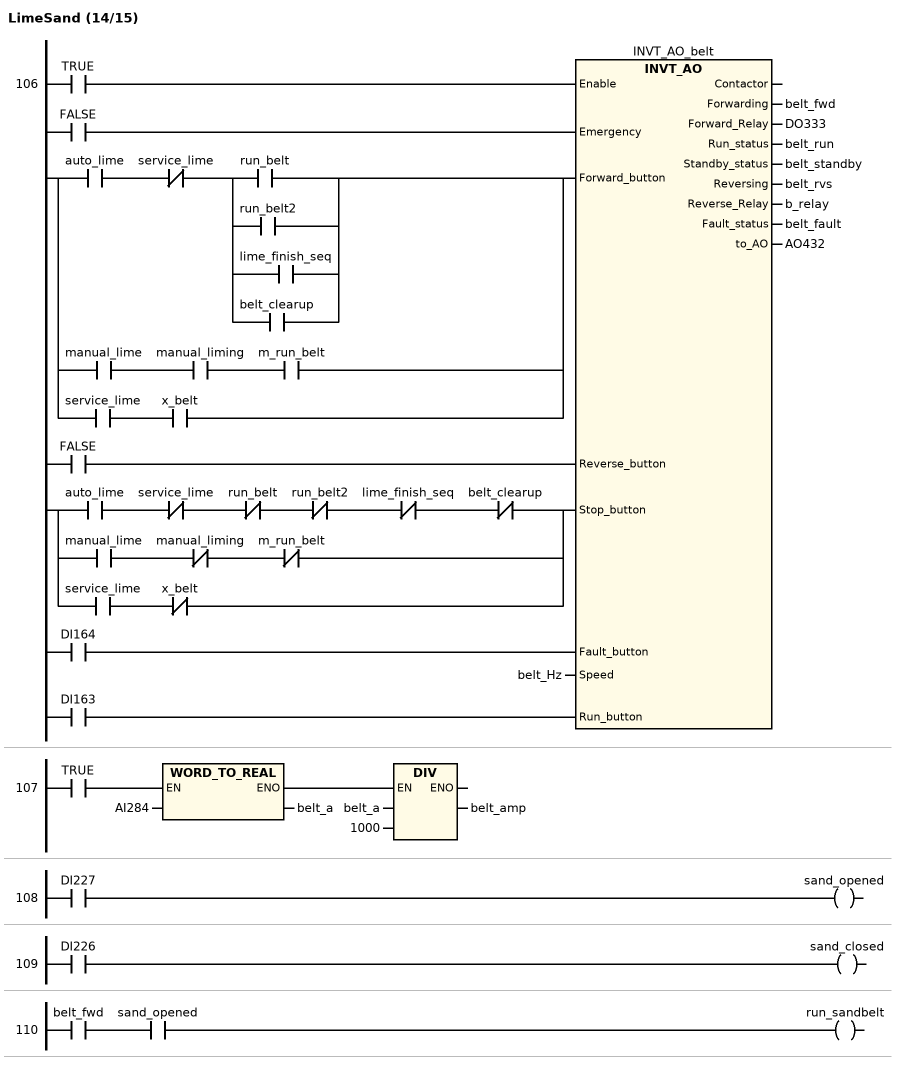
// NETWORK 106
INVT_AO_belt(
    Enable := TRUE,
    Emergency := FALSE,
    Forward_button := auto_lime AND NOT service_lime AND (run_belt OR run_belt2 OR lime_finish_seq OR belt_clearup) OR manual_lime AND manual_liming AND m_run_belt OR service_lime AND x_belt,
    Reverse_button := FALSE,
    Stop_button := auto_lime AND NOT service_lime AND NOT run_belt AND NOT run_belt2 AND NOT lime_finish_seq AND NOT belt_clearup OR manual_lime AND NOT manual_liming AND NOT m_run_belt OR service_lime AND NOT x_belt,
    Fault_button := DI164,
    Speed := belt_Hz,
    Run_button := DI163,
    Forwarding => belt_fwd,
    Forward_Relay => DO333,
    Run_status => belt_run,
    Standby_status => belt_standby,
    Reversing => belt_rvs,
    Reverse_Relay => b_relay,
    Fault_status => belt_fault,
    to_AO => AO432); // INVT_AO

// NETWORK 107
belt_a := WORD_TO_REAL(AI284);
belt_amp := belt_a / 1000;

// NETWORK 108
sand_opened := DI227;

// NETWORK 109
sand_closed := DI226;

// NETWORK 110
run_sandbelt := belt_fwd AND sand_opened;

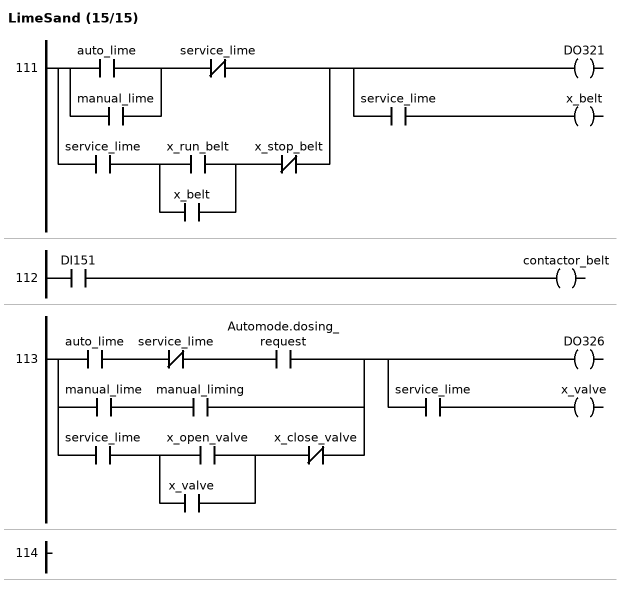
// NETWORK 111
_w14 := (auto_lime OR manual_lime) AND NOT service_lime OR service_lime AND (x_run_belt OR x_belt) AND NOT x_stop_belt;
DO321 := _w14;
x_belt := _w14 AND service_lime;

// NETWORK 112
contactor_belt := DI151;

// NETWORK 113
_w15 := auto_lime AND NOT service_lime AND Automode.dosing_request OR manual_lime AND manual_liming OR service_lime AND (x_open_valve OR x_valve) AND NOT x_close_valve;
DO326 := _w15;
x_valve := _w15 AND service_lime;

// NETWORK 114

END_PROGRAM

// Device/Application/BAYKON
FUNCTION_BLOCK BAYKON
VAR_INPUT
	stat: WORD;
	REG07: WORD;
END_VAR
VAR
	weight_real: REAL;
	weight_signature: REAL;
	positive_w: BOOL;
	weight_realx: REAL;
	weight_realm: REAL;
END_VAR
VAR_OUTPUT
	fault_info: STRING;
	system_info: STRING;
	data_info: STRING;
END_VAR
VAR_INPUT
	REG06: WORD;
END_VAR
VAR_OUTPUT
	weight: REAL;
END_VAR
VAR
	No_Error: BOOL;
END_VAR
VAR
	ADC_out_of_range: BOOL;
	ADC_over_range: BOOL;
	ADC_under_range: BOOL;
	System_error: BOOL;
	IN_programing_mode: BOOL;
	Low_or_high_voltage_det: BOOL;
END_VAR
VAR_INPUT
	Enable: BOOL;
END_VAR

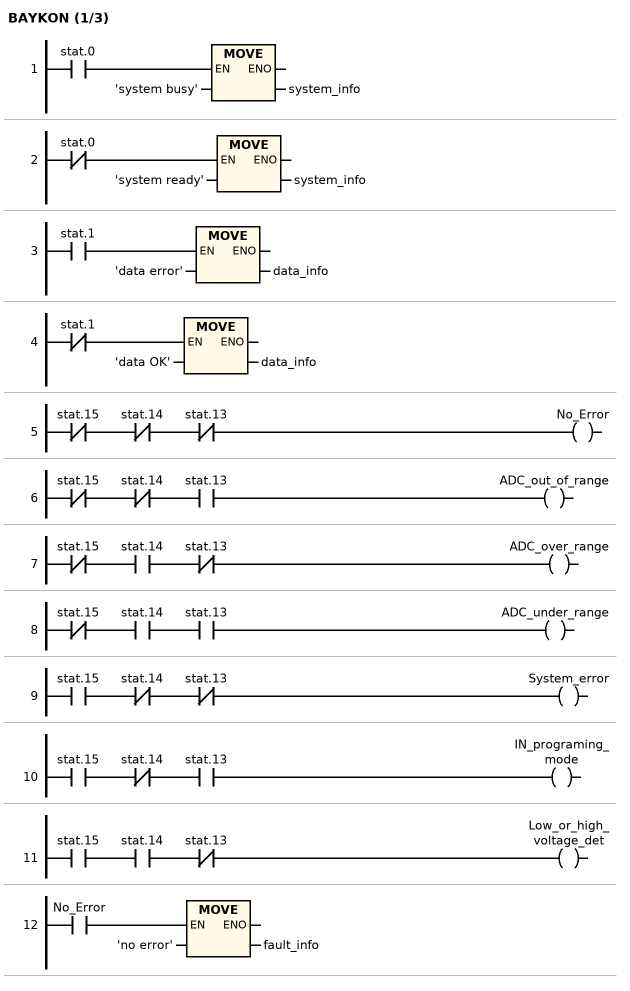
// NETWORK 1
IF stat.0 THEN system_info := 'system busy'; END_IF

// NETWORK 2
IF NOT stat.0 THEN system_info := 'system ready'; END_IF

// NETWORK 3
IF stat.1 THEN data_info := 'data error'; END_IF

// NETWORK 4
IF NOT stat.1 THEN data_info := 'data OK'; END_IF

// NETWORK 5
No_Error := NOT stat.15 AND NOT stat.14 AND NOT stat.13;

// NETWORK 6
ADC_out_of_range := NOT stat.15 AND NOT stat.14 AND stat.13;

// NETWORK 7
ADC_over_range := NOT stat.15 AND stat.14 AND NOT stat.13;

// NETWORK 8
ADC_under_range := NOT stat.15 AND stat.14 AND stat.13;

// NETWORK 9
System_error := stat.15 AND NOT stat.14 AND NOT stat.13;

// NETWORK 10
IN_programing_mode := stat.15 AND NOT stat.14 AND stat.13;

// NETWORK 11
Low_or_high_voltage_det := stat.15 AND stat.14 AND NOT stat.13;

// NETWORK 12
IF No_Error THEN fault_info := 'no error'; END_IF

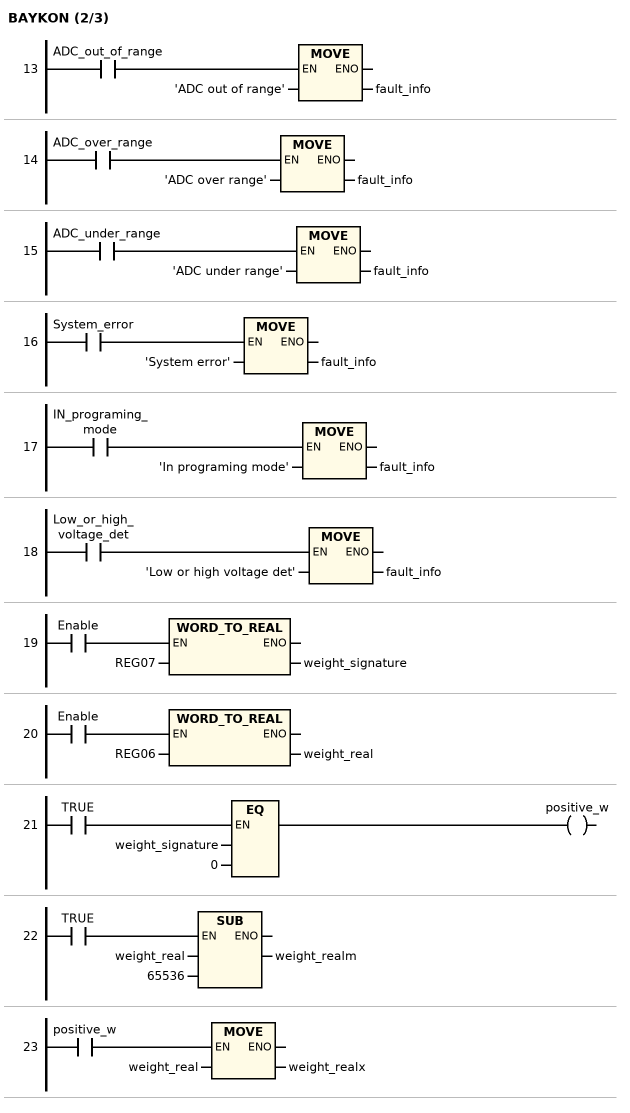
// NETWORK 13
IF ADC_out_of_range THEN fault_info := 'ADC out of range'; END_IF

// NETWORK 14
IF ADC_over_range THEN fault_info := 'ADC over range'; END_IF

// NETWORK 15
IF ADC_under_range THEN fault_info := 'ADC under range'; END_IF

// NETWORK 16
IF System_error THEN fault_info := 'System error'; END_IF

// NETWORK 17
IF IN_programing_mode THEN fault_info := 'In programing mode'; END_IF

// NETWORK 18
IF Low_or_high_voltage_det THEN fault_info := 'Low or high voltage det'; END_IF

// NETWORK 19
IF Enable THEN weight_signature := WORD_TO_REAL(REG07); END_IF

// NETWORK 20
IF Enable THEN weight_real := WORD_TO_REAL(REG06); END_IF

// NETWORK 21
positive_w := weight_signature = 0;

// NETWORK 22
weight_realm := weight_real - 65536;

// NETWORK 23
IF positive_w THEN weight_realx := weight_real; END_IF

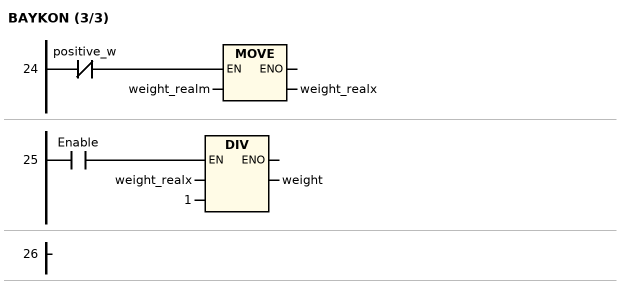
// NETWORK 24
IF NOT positive_w THEN weight_realx := weight_realm; END_IF

// NETWORK 25
IF Enable THEN weight := weight_realx / 1; END_IF

// NETWORK 26

END_FUNCTION_BLOCK

// Device/Application/screw_speed
FUNCTION_BLOCK screw_speed
VAR_INPUT
	enable: BOOL;
	starting_weight: REAL;
END_VAR
VAR
	target_per: REAL;
END_VAR
VAR_INPUT
	weight_in: REAL;
	target_weight: REAL := 1;
	slow_set: REAL := 70;
END_VAR
VAR_OUTPUT
	target_fix: REAL;
	speed: REAL;
END_VAR
VAR_INPUT
	max_speed: REAL;
END_VAR
VAR
	speed_adj_range: REAL;
END_VAR
VAR_INPUT
	min_speed: REAL;
END_VAR
VAR
	weight_onslow: REAL;
	slow_per: REAL;
	slow_speed: REAL;
END_VAR
VAR_INPUT
	slow_set2: REAL := 95;
END_VAR

IF enable = TRUE THEN
	target_fix := target_weight + starting_weight;
	target_per := (weight_in / target_fix) *100;
	speed_adj_range := max_speed - min_speed;
	weight_onslow := target_fix * ((100 - slow_set)/100);
	slow_per := ((target_fix - weight_in)/weight_onslow)*100;
	slow_speed := (slow_per * speed_adj_range) + min_speed; 
	IF target_per <= slow_set THEN
		speed := max_speed;
	END_IF
	IF target_per > slow_set AND target_per < slow_set2 THEN
		speed := slow_speed/100;
	END_IF
	IF target_per >= slow_set2 THEN
		speed := min_speed;
	END_IF
	ELSE
		speed := 0;
END_IF

END_FUNCTION_BLOCK

// Device/Application/INVT_AO
FUNCTION_BLOCK INVT_AO
VAR_INPUT
	Enable: BOOL;
	Emergency: BOOL;
	Forward_button: BOOL;
	Reverse_button: BOOL;
	Stop_button: BOOL;
	Fault_button: BOOL;
	// input in Hz*100 (5000 for 50Hz)
	Speed: REAL;
	
	Run_button: BOOL;
END_VAR
VAR_OUTPUT
	Contactor: BOOL;
	Forwarding: BOOL;
	Forward_Relay: BOOL;
	Run_status: BOOL;
END_VAR
VAR
	Interuprt: BOOL;
	Real_value: REAL;
	AO_real: REAL;
END_VAR
VAR_OUTPUT
	Standby_status: BOOL;
	Reversing: BOOL;
	Reverse_Relay: BOOL;
	Fault_status: BOOL;
	to_AO: WORD;
END_VAR

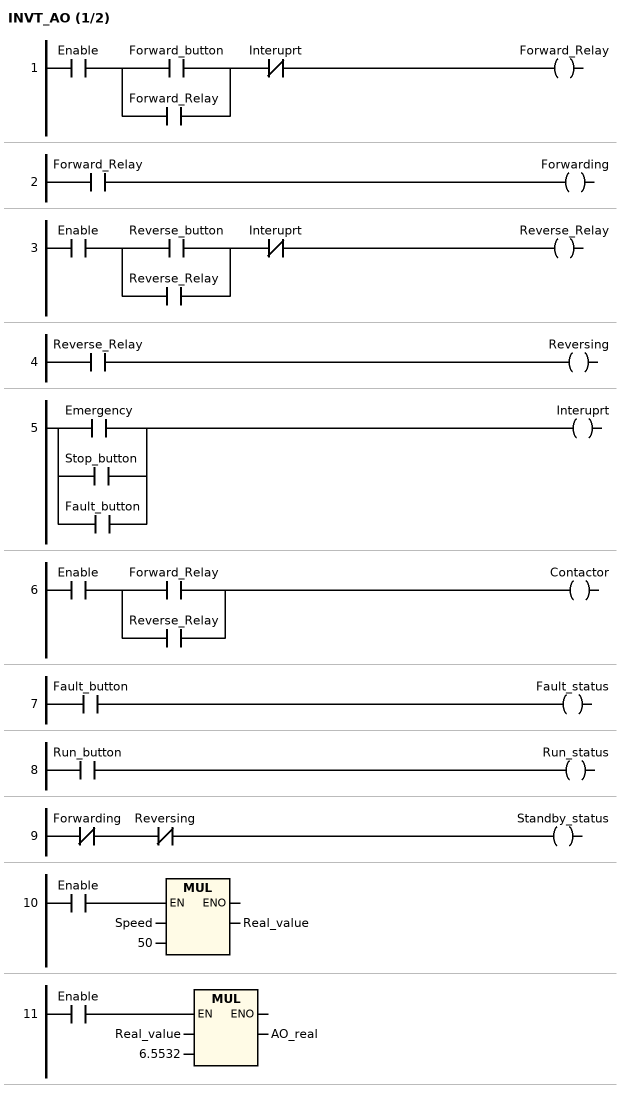
// NETWORK 1
Forward_Relay := Enable AND (Forward_button OR Forward_Relay) AND NOT Interuprt;

// NETWORK 2
Forwarding := Forward_Relay;

// NETWORK 3
Reverse_Relay := Enable AND (Reverse_button OR Reverse_Relay) AND NOT Interuprt;

// NETWORK 4
Reversing := Reverse_Relay;

// NETWORK 5
Interuprt := Emergency OR Stop_button OR Fault_button;

// NETWORK 6
Contactor := Enable AND (Forward_Relay OR Reverse_Relay);

// NETWORK 7
Fault_status := Fault_button;

// NETWORK 8
Run_status := Run_button;

// NETWORK 9
Standby_status := NOT Forwarding AND NOT Reversing;

// NETWORK 10
IF Enable THEN Real_value := Speed * 50; END_IF

// NETWORK 11
IF Enable THEN AO_real := Real_value * 6.5532; END_IF

